// TIA Portal V20 export
TYPE "LKinCtrl_typeCOffPathDataOut"
   STRUCT
      nextCommand : "LKinCtrl_typePathDataElement";   // Target data - next command
      intermediateCommand : "LKinCtrl_typePathDataElement";   // Target data - intermediate (additional) command
      nextButOneCommand : "LKinCtrl_typeCOffOutNextButOneCmd";   // Target data - next but one command
      nextPositionAbsolute : "LKinCtrl_typeCartesianPosition";   // Source data - next absolute position
      nextPositionAbsoluteRadComp : "LKinCtrl_typeCartesianPosition";   // Source data - next absolute position (radius compensated)
   END_STRUCT;
   // nextCommand.cmdParameters.transitionParameters[1] := -1.0;
   // intermediateCommand.cmdParameters.transitionParameters[1] := -1.0;
END_TYPE
